PROGRAM Axis02_Alarm
VAR
	Always_ON	:	BOOL	:=TRUE	;//상시 ON 
	Always_OFF	:	BOOL	:=FALSE	;//상시 OFF
END_VAR

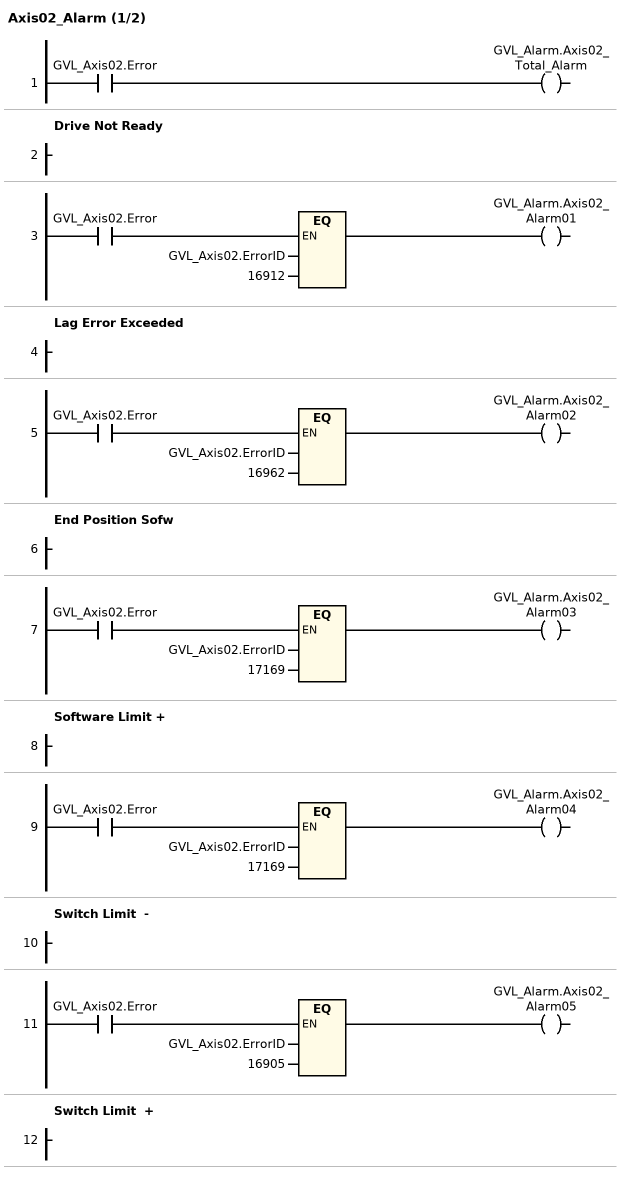
// NETWORK 1
GVL_Alarm.Axis02_Total_Alarm := GVL_Axis02.Error;

// NETWORK 2: Drive Not Ready

// NETWORK 3
GVL_Alarm.Axis02_Alarm01 := GVL_Axis02.Error AND GVL_Axis02.ErrorID = 16912;

// NETWORK 4: Lag Error Exceeded

// NETWORK 5
GVL_Alarm.Axis02_Alarm02 := GVL_Axis02.Error AND GVL_Axis02.ErrorID = 16962;

// NETWORK 6: End Position Sofw

// NETWORK 7
GVL_Alarm.Axis02_Alarm03 := GVL_Axis02.Error AND GVL_Axis02.ErrorID = 17169;

// NETWORK 8: Software Limit +

// NETWORK 9
GVL_Alarm.Axis02_Alarm04 := GVL_Axis02.Error AND GVL_Axis02.ErrorID = 17169;

// NETWORK 10: Switch Limit -

// NETWORK 11
GVL_Alarm.Axis02_Alarm05 := GVL_Axis02.Error AND GVL_Axis02.ErrorID = 16905;

// NETWORK 12: Switch Limit +

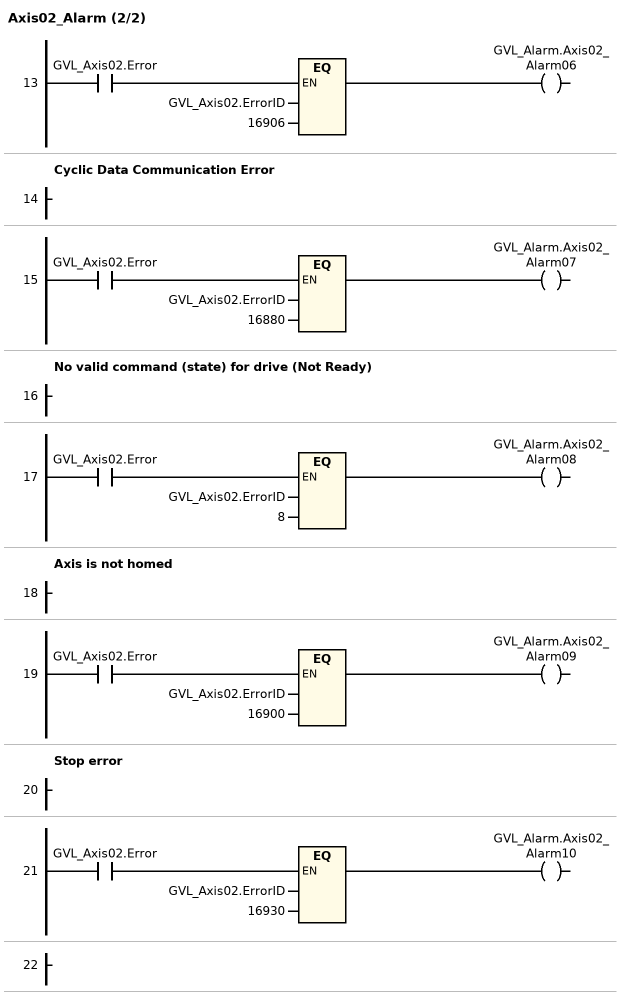
// NETWORK 13
GVL_Alarm.Axis02_Alarm06 := GVL_Axis02.Error AND GVL_Axis02.ErrorID = 16906;

// NETWORK 14: Cyclic Data Communication Error

// NETWORK 15
GVL_Alarm.Axis02_Alarm07 := GVL_Axis02.Error AND GVL_Axis02.ErrorID = 16880;

// NETWORK 16: No valid command (state) for drive (Not Ready)

// NETWORK 17
GVL_Alarm.Axis02_Alarm08 := GVL_Axis02.Error AND GVL_Axis02.ErrorID = 8;

// NETWORK 18: Axis is not homed

// NETWORK 19
GVL_Alarm.Axis02_Alarm09 := GVL_Axis02.Error AND GVL_Axis02.ErrorID = 16900;

// NETWORK 20: Stop error

// NETWORK 21
GVL_Alarm.Axis02_Alarm10 := GVL_Axis02.Error AND GVL_Axis02.ErrorID = 16930;

// NETWORK 22

END_PROGRAM

(* stored: Version 1.1.0.1, ProductVersion 3.1.4024.15
   POU Axis02_Alarm: Id {f6f9ac42-b997-434b-b5a4-9eb789bbb771}, SpecialFunc None *)
